// TwinCAT 3 PLC project EventLogger
// ProgramVersion: 3.1.4026.1+972e9c44872ad038b353624a861fd7e3244e9f75
// libraries:
//   Anker Andersen Library, * (AnkerAndersen A_S)
//   Tc2_Standard, * (Beckhoff Automation GmbH)
//   Tc2_System, * (Beckhoff Automation GmbH)
//   Tc2_Utilities, * (Beckhoff Automation GmbH)
// project tree:
//   DUTs/ E_EventType.TcDUT (not stored), ST_Event.TcDUT (not stored)
//   / PlcTask.TcTTO
//   POUs/ FB_EventBuffer.TcPOU (not stored), FB_EventLogger.TcPOU (not stored), FB_CsvPersistantEventStorage.TcPOU (not stored), F_UpdateEventTimestampWithSystemTime.TcPOU (not stored), I_PersistantEventStorage.TcIO, MAIN.TcPOU
// real-time tasks:
//   TASK PlcTask: cycle T#10ms, priority 20, ADS port 350

CONFIGURATION EventLogger
    RESOURCE PLC ON TwinCAT3
        TASK PlcTask(INTERVAL := T#10ms, PRIORITY := 20);
        PROGRAM MAIN WITH PlcTask : MAIN;
    END_RESOURCE
END_CONFIGURATION

// ---- POUs/I_PersistantEventStorage.TcIO
INTERFACE  I_PersistantEventStorage

METHOD M_StoreEvent
VAR_INPUT
	stEvent : ST_Event;
END_VAR
END_METHOD

END_INTERFACE

// ---- POUs/MAIN.TcPOU
PROGRAM MAIN
VAR
END_VAR

END_PROGRAM
